// TIA Portal V19 export
DATA_BLOCK "MODE SELECTION DB"   // DB3
{ S7_Optimized_Access := 'FALSE' }
   VAR
      "RO-1" : Struct
         AUTO : Bool;
         MANUAL : Bool;
         STANDBY : Bool;
         "MODE BUFF" : Int;
         "PROCESS BUFF" : Int;
         START : Bool;
         STOP : Bool;
      END_STRUCT;
      "RO-2" : Struct
         AUTO : Bool;
         MANUAL : Bool;
         STANDBY : Bool;
         "MODE BUFF" : Int;
         "PROCESS BUFF" : Int;
         START : Bool;
         STOP : Bool;
      END_STRUCT;
      EDI : Struct
         AUTO : Bool;
         MANUAL : Bool;
         STANDBY : Bool;
         "MODE BUFF" : Int;
         "PROCESS BUFF" : Int;
         START : Bool;
         STOP : Bool;
      END_STRUCT;
   END_VAR
BEGIN
END_DATA_BLOCK
